// TIA Portal V20 export
// export: Created 2025-12-01T14:57:43.8043943Z, ExportSetting None, DisplayName Totally Integrated Automation Portal, DisplayVersion V20 Update 3, DisplayName TIA Portal Openness, DisplayVersion V20 Update 3, DisplayName TIA Portal Version Control Interface, DisplayVersion V20 Update 3, DisplayName STEP 7 Professional, DisplayVersion V20 Update 3, DisplayName STEP 7 Safety, DisplayVersion V20 Update 2, DisplayName WinCC Basic/Comfort/Advanced, DisplayVersion V20 Update 3, DisplayName WinCC Professional, DisplayVersion V20 Update 3, DisplayName WinCC Unified, DisplayVersion V20 Update 3
FUNCTION "FC513_TL_Etiqueta_EnMesaCruce_ULINT" : Void   // FC513, LAD
{ S7_Optimized_Access := 'FALSE' }
// stored: AutoNumber false, SetENOAutomatically false
   VAR_INPUT
      Mesa : UInt;   // Numero de Mesa CON OFFSET
      Mesa_S01 : UInt;   // Mesa de Salida por S01 CON OFFSET
      Mesa_S02 : UInt;   // Mesa de Salida por S02 CON OFFSET
      Mesa_S03 : UInt;   // Mesa de Salida por S03 CON OFFSET
      Mesa_S04 : UInt;   // Mesa de Salida por S04 CON OFFSET
      Etiqueta : ULInt;   // Etiqueta
      OrdenEjecutada : UInt;   // Orden Ejecutada en el Cruce
      MesaDeJDT02 : Bool;
   END_VAR
   VAR_TEMP
      MesaTMP : UDInt;
      MotivoTMP : UDInt;
      Posicion : Int;
      i : Int;
      longitud : Int;
      string_motivo : String[10];
      string_mesa : String[12];
      codigo_string : String[20];
   END_VAR
BEGIN

REGION Network 1 (SCL)
   //---------------------------------------------------------------------------------------------
   // --- 
   // --- Condiciones para enviar el Nuevo Evento
   // ---     Cerrado el Protocolo de la Mesa
   // --- Recoger - Presencias de la Mesa
   // --- Emitiendo Mensajes
   // ---
   // ---------------------------------------------------------------------------------------------
   // ------- Cerrado el Protocolo de la Mesa
   // 
   IF "DB810_ColasMesas".Colas[#Mesa].EstadoPresenciaMesa <> 0 THEN
       RETURN;
   END_IF;


   // ---------------------------------------------------------------------------------------------
   // ------- Recoger - Presencias de la Mesa
   // ---------------------------------------------------------------------------------------------

   IF "DB840_Emision".Mesa[#Mesa].Protocolo.PresRouter = FALSE THEN
       RETURN;
   END_IF;

   // ---------------------------------------------------------------------------------------------
   // ------- Recoger Datos para la Generacion del Evento

   #MotivoTMP := #OrdenEjecutada / 10;
   #MesaTMP := #OrdenEjecutada MOD 10;
END_REGION

REGION Network 2 (SCL)
   // miramos si tenemos hueco para emitir hacia el jdt que nos corresponde
   // 
   IF #MesaDeJDT02=true THEN
       REGION buscar en JDT2

           #Posicion := -1;
           FOR #i := 0 TO 100 BY 1 DO
               #longitud := LEN("DB197_eventos_generados_routing_JDT2".evento[#i]);
               IF #longitud = 0 THEN
                   #Posicion := #i;
                   EXIT;
               END_IF;
           END_FOR;

           // si no hay sitio para escribir salimos del bloque
           IF #Posicion = -1 THEN
               RETURN;
           END_IF;
       END_REGION
       ;
   ELSE
       REGION buscar en JDT1

           #Posicion := -1;
           FOR #i := 0 TO 100 BY 1 DO
               #longitud := LEN("DB198_eventos_generados_routing_JDT1".evento[#i]);
               IF #longitud = 0 THEN
                   #Posicion := #i;
                   EXIT;
               END_IF;
           END_FOR;

           // si no hay sitio para escribir salimos del bloque
           IF #Posicion = -1 THEN
               RETURN;
           END_IF;
       END_REGION
   END_IF;
END_REGION

REGION Network 3 (SCL)

   CASE #MotivoTMP OF
       0:
           #string_motivo := '[MOTI]NORM';         // --- Escribir - Motivo NORMAL  (0)
       1:
           #string_motivo := '[MOTI]BLOQ';     // --- Escribir - Motivo BLOQUEO (1)
       2:
           #string_motivo := '[MOTI]VACI';   // --- Escribir - Motivo VACIADO (2)
       3:
           #string_motivo := '[MOTI]ERRO';  // --- Escribir - Motivo ETIQUETA ERROR (3)
       4:
           #string_motivo := '[MOTI]NENC';// --- Escribir - Motivo ETIQUETA NO ENCONTRADA (4)
       5:
           #string_motivo := '[MOTI]INIC'; // --- Escribir - Motivo Ejecucion por INICIALIZACION (5)
       6:
           #string_motivo := '[MOTI]XJDT';// --- Escribir - Motivo Ejecucion por JDT (6)
       7:
           #string_motivo := '[MOTI]BLKC';  // --- Escribir - Motivo Ejecucion por Bloqueo intentando Continuar (7)
       8:
           #string_motivo := '[MOTI]BLKE'; // --- Escribir - Motivo Ejecucion por Bloqueo intentando Entrar (8)


       ELSE
           #string_motivo := '[MOTI]DESC';

   END_CASE;

   CASE #MesaTMP OF

       1:
           #string_mesa := CONCAT(IN1 := '[MESA]', IN2 := DELETE(IN := (UDINT_TO_STRING(IN := #Mesa_S01)), L := 1, P := 1));
       2:
           #string_mesa := CONCAT(IN1 := '[MESA]', IN2 := DELETE(IN := (UDINT_TO_STRING(IN := #Mesa_S02)), L := 1, P := 1));
       3:
           #string_mesa := CONCAT(IN1 := '[MESA]', IN2 := DELETE(IN := (UDINT_TO_STRING(IN := #Mesa_S03)), L := 1, P := 1));
       4:
           #string_mesa := CONCAT(IN1 := '[MESA]', IN2 := DELETE(IN := (UDINT_TO_STRING(IN := #Mesa_S04 )), L := 1, P := 1));

       ELSE  // Statement section ELSE
           #string_mesa := CONCAT(IN1 := '[MESA]', IN2 := DELETE(IN := (UDINT_TO_STRING(IN := #Mesa)), L := 1, P := 1));

   END_CASE;

   #codigo_string := DELETE(IN := (ULINT_TO_STRING(IN :=#Etiqueta)), L := 1, P := 1);


   IF #MesaDeJDT02 = true THEN

       "DB197_eventos_generados_routing_JDT2".evento[#Posicion] := CONCAT(IN1 := '{PRES', IN2 := #string_mesa, IN3 := '[SSCC]', IN4 := #codigo_string, IN5 := #string_motivo, IN6 := "DB921_DATOS_FECHA_HORA".TIME_STAMP, IN7:='}');

   ELSE
       "DB198_eventos_generados_routing_JDT1".evento[#Posicion] := CONCAT(IN1 := '{PRES', IN2 := #string_mesa, IN3 := '[SSCC]', IN4 := #codigo_string, IN5 := #string_motivo, IN6 := "DB921_DATOS_FECHA_HORA".TIME_STAMP, IN7:='}');

   END_IF;

   "DB841_Recepcion".Mesa[#Mesa].Protocolo.EmiOK := TRUE;
   "DB810_ColasMesas".Colas[#Mesa].EstadoPresenciaMesa := 1;
END_REGION
END_FUNCTION
